TYPE EtcMasterBase_62654B43 :
STRUCT
END_STRUCT
END_TYPE

(* stored: Version 1.2.0.0, ProductVersion 3.1.4024.11
   DUT EtcMasterBase_62654B43: Id {6a095e8b-a034-4d38-8b33-d0ab19db4210} *)
